FUNCTION_BLOCK Test_TStreamAdd_Read_BLOB EXTENDS T_UnitTestBase
VAR
    Stream : T_Stream(StreamLength := 2);
    Now    : TIMESTRUCT := (wDay := 23,
            wMonth := 12,
            wYear := 1945,
            wHour := 22,
            wMinute := 20,
            wSecond := 18);
    NowFromStream : TIMESTRUCT;

    LREAL_Value : LREAL := 1.234;
END_VAR

Stream.Init(2);
NowFromStream.wDay    := 0;
NowFromStream.wMonth  := 0;
NowFromStream.wYear   := 0;
NowFromStream.wHour   := 0;
NowFromStream.wMinute := 0;
NowFromStream.wSecond := 0;

Stream.SetNextArgTypeId(E_ArgTypeId.Type_Blob);
Stream.Add_BLOB(Now);

Stream.Seek(0);

IF Stream.GetNextArgTypeId() = E_ArgTypeId.Type_Blob THEN
    Stream.Read_BLOB(NowFromStream);
END_IF

// check the value...
Assertion.AssertEquals_BLOB(Expected     := Now,
                            Actual       := NowFromStream,
                            VariableName := 'NowFromStream');

// check we are at the end of the stream..							
Assertion.AssertEquals_UDINT(Expected     := Stream.StreamLength,
                             Actual       := Stream.Position,
                             VariableName := 'Stream.Position');

TestFinished();

END_FUNCTION_BLOCK

(* stored: Version 1.1.0.1, ProductVersion 3.1.4024.6
   POU Test_TStreamAdd_Read_BLOB: Id {c3912488-96c9-4cb9-bb2e-8d80ca1f3426}, SpecialFunc None *)
